TYPE ST_StateMachine_State :
STRUCT
	nState	: INT;
	sState	: STRING;
END_STRUCT
END_TYPE

(* stored: Version 1.1.0.1, ProductVersion 3.1.4026.18
   DUT ST_StateMachine_State: Id {9b470c85-e673-4fff-a5ed-92c7c0a9296c} *)
